Yaskawa INFORM job: X2_104(180,0).JBI

/JOB
//NAME X2_104(180,0)
//POS
///NPOS 390,390,390,11,0,0
///TOOL 0
///POSTYPE PULSE
///PULSE
C00000=2822,-118876,-115474,-188,81202,276
C00001=-104800,-59825,-68378,-15730,82561,27134
C00002=-104796,-59871,-65452,-15790,80804,27361
C00003=-104795,-59835,-64253,-15818,80110,27451
C00004=-104794,-59728,-62536,-15861,79145,27577
C00005=-104795,-59835,-64253,-15818,80110,27451
C00006=-104795,-59821,-63969,-15825,79949,27472
C00007=-104795,-59821,-63967,-15825,79948,27473
C00008=-104795,-59821,-63969,-15825,79949,27472
C00009=-104795,-59821,-63969,-15825,79949,27472
C00010=-104794,-59750,-62822,-15854,79304,27557
C00011=-104793,-59760,-62819,-15854,79297,27558
C00012=-104794,-59750,-62822,-15854,79304,27557
C00013=-104795,-59822,-63970,-15825,79949,27472
C00014=-104795,-59835,-64253,-15818,80110,27451
C00015=-104796,-59871,-65452,-15790,80804,27361
C00016=-104800,-59825,-68378,-15730,82561,27134
C00017=-108679,-64626,-75582,-9628,93281,21595
C00018=-143431,-69229,-73342,20821,87037,-27373
C00019=-148549,-57792,-61137,30779,82601,-29503
C00020=-148549,-57540,-58627,30861,81376,-29834
C00021=-148549,-57408,-57604,30899,80891,-29966
C00022=-148550,-57145,-55796,30970,80047,-30197
C00023=-148549,-57408,-57604,30899,80891,-29966
C00024=-149525,-56700,-57014,31060,81250,-30254
C00025=-148546,-57369,-57388,30906,80793,-29992
C00026=-148548,-57377,-57384,30907,80788,-29994
C00027=-148549,-57379,-57388,30907,80789,-29994
C00028=-148544,-57403,-57724,30893,80955,-29947
C00029=-148544,-57403,-57721,30893,80954,-29947
C00030=-148544,-57403,-57724,30893,80955,-29947
C00031=-148549,-57379,-57388,30907,80789,-29994
C00032=-148549,-57408,-57604,30899,80891,-29966
C00033=-148549,-57540,-58627,30861,81376,-29834
C00034=-148549,-57792,-61137,30779,82601,-29503
C00035=-143431,-69229,-73342,20821,87037,-27373
C00036=-113515,-83541,-80276,-7171,73507,8599
C00037=-114214,-69268,-73638,-6873,76673,8174
C00038=-114213,-69131,-70631,-6922,74904,8274
C00039=-114212,-69024,-69400,-6944,74207,8314
C00040=-114212,-68820,-67637,-6976,73234,8370
C00041=-114212,-69024,-69400,-6944,74207,8314
C00042=-114212,-68905,-68252,-6965,73567,8351
C00043=-114211,-68906,-68249,-6965,73564,8351
C00044=-114212,-68905,-68252,-6965,73567,8351
C00045=-114212,-69039,-69496,-6942,74258,8311
C00046=-114213,-69247,-72540,-6890,76013,8211
C00047=-113515,-83541,-80276,-7171,73507,8599
C00048=-121193,-82756,-80438,381,72886,-91
C00049=-121146,-70418,-74709,362,75701,-66
C00050=-121146,-70284,-71707,364,73922,-71
C00051=-121146,-70176,-70478,365,73221,-73
C00052=-121145,-69975,-68718,367,72241,-76
C00053=-121146,-70176,-70478,365,73221,-73
C00054=-121145,-70029,-69144,367,72475,-75
C00055=-121145,-70029,-69141,367,72474,-75
C00056=-121145,-70029,-69144,367,72475,-75
C00057=-121152,-71796,-70447,369,72370,-78
C00058=-124110,-69926,-69074,1277,72515,-1113
C00059=-138593,-60519,-63927,18922,79598,-16349
C00060=-137648,-60917,-64139,18714,79312,-16056
C00061=-140210,-64003,-66362,19292,79697,-16914
C00062=-130105,-77106,-75700,9072,74443,-7764
C00063=-121203,-87562,-80341,388,70357,-102
C00064=-121146,-70284,-71707,364,73922,-71
C00065=-121146,-70418,-74709,362,75701,-66
C00066=-121193,-82756,-80438,381,72886,-91
C00067=-119439,-80664,-79685,-1380,73580,1904
C00068=-119526,-70071,-74713,-1339,75962,1848
C00069=-119525,-69957,-71718,-1350,74178,1867
C00070=-119525,-69858,-70493,-1354,73475,1875
C00071=-119525,-69668,-68738,-1361,72493,1886
C00072=-119525,-69858,-70493,-1354,73475,1875
C00073=-119525,-69702,-69020,-1360,72649,1884
C00074=-119525,-69702,-69016,-1360,72646,1885
C00075=-119525,-69702,-69020,-1360,72649,1884
C00076=-119525,-69851,-70308,-1355,73364,1876
C00077=-120731,-69912,-70673,-987,73540,1455
C00078=-119525,-69885,-70669,-1354,73569,1874
C00079=-119525,-69895,-70665,-1354,73562,1874
C00080=-119525,-69721,-69012,-1360,72634,1885
C00081=-119525,-69858,-70493,-1354,73475,1875
C00082=-119525,-69957,-71718,-1350,74178,1867
C00083=-119526,-70071,-74713,-1339,75962,1848
C00084=-108249,-94324,-77488,56,64739,4382
C00085=-108596,-86932,-71529,170,64871,4253
C00086=-108725,-84070,-69130,212,64865,4205
C00087=-105542,-82906,-68648,-826,65188,5383
C00088=-119360,-76750,-65885,13584,70522,-11705
C00089=-122073,-72654,-64134,16061,73903,-15414
C00090=-121979,-72766,-64187,16042,73861,-15386
C00091=-122522,-71846,-63747,16636,74615,-16299
C00092=-129432,-59927,-56905,23211,83184,-32001
C00093=-127456,-72696,-62533,22682,75276,-32884
C00094=-129013,-74086,-64315,22925,76062,-33315
C00095=-132460,-77476,-68693,23432,77911,-34241
C00096=-135381,-103003,-79022,24540,72556,-36456
C00097=-155606,-83763,-70294,33424,82257,-10320
C00098=-151405,-68724,-63344,32871,83525,-8251
C00099=-152125,-66994,-60639,32982,83150,-8650
C00100=-148800,-61641,-56056,32604,81881,-7710
C00101=-126757,-81773,-69022,8384,64119,9204
C00102=-127031,-82170,-69267,3063,63090,13556
C00103=-124915,-87939,-73263,2287,62515,14340
C00104=-115381,-93439,-79772,-9030,66985,13175
C00105=-91545,-88698,-72787,-32521,79113,9069
C00106=-71683,-72063,-68966,-26106,87557,15526
C00107=-79934,-51849,-58812,-25261,88765,12201
C00108=-82185,-48076,-53683,-24983,86983,11751
C00109=-83735,-47880,-52547,-24792,85977,11391
C00110=-84464,-48873,-53018,-24699,85557,11210
C00111=-94891,-61855,-60139,-23205,80447,8398
C00112=-100780,-70938,-64689,-19538,73748,2674
C00113=-115179,-76942,-67444,-14121,68125,-4118
C00114=-111498,-78431,-66563,-20592,66506,-6661
C00115=-124355,-85604,-69411,-6892,57492,-20990
C00116=-144608,-76157,-64843,18668,63245,-44599
C00117=-155294,-46121,-48462,31776,84228,-61563
C00118=-157048,-60165,-52454,36767,71330,-65698
C00119=-158808,-60243,-53717,36995,72681,-65990
C00120=-162225,-60657,-56708,37410,75470,-66490
C00121=-167417,-72784,-64632,35375,81907,-66933
C00122=-116272,-113725,-85439,-7807,65506,33606
C00123=-117374,-79868,-72519,-7126,74775,32629
C00124=-119711,-75631,-67242,-6610,73513,31878
C00125=-120783,-73750,-64961,-6368,72993,31529
C00126=-120584,-71036,-63698,-6398,73621,31564
C00127=-120975,-79246,-65174,-5752,61943,44903
C00128=-119928,-81186,-67588,-6116,62507,45272
C00129=-117420,-85347,-72820,-6980,63787,46146
C00130=-116281,-118301,-84670,-8155,54332,47249
C00131=846,-162146,-127518,2443,90805,10094
C00132=846,-162146,-127518,2443,90805,10094
C00133=-127354,-61380,-68788,13702,79975,-24096
C00134=-125311,-61634,-65992,13253,77838,-23621
C00135=-124491,-61652,-64830,13073,76999,-23425
C00136=-124495,-61511,-63095,13123,76029,-23531
C00137=-124491,-61652,-64830,13073,76999,-23425
C00138=-124521,-61630,-64544,13089,76844,-23452
C00139=-124525,-61630,-64553,13090,76850,-23453
C00140=-124521,-61630,-64544,13089,76844,-23452
C00141=-124480,-61634,-64545,13078,76835,-23439
C00142=-124482,-61539,-63385,13111,76187,-23509
C00143=-122660,-61663,-63447,12634,75875,-22900
C00144=-124482,-61539,-63385,13111,76187,-23509
C00145=-124480,-61634,-64545,13078,76835,-23439
C00146=-124491,-61652,-64830,13073,76999,-23425
C00147=-125311,-61634,-65992,13253,77838,-23621
C00148=-127354,-61380,-68788,13702,79975,-24096
C00149=-122646,-60819,-73208,8582,92262,-18154
C00150=-97025,-77240,-76763,-20966,85097,28182
C00151=-93139,-57918,-60776,-30781,82021,29693
C00152=-93133,-57672,-58277,-30872,80802,30026
C00153=-93131,-57543,-57259,-30912,80319,30159
C00154=-93129,-57265,-55441,-30989,79477,30390
C00155=-93131,-57543,-57259,-30912,80319,30159
C00156=-93130,-57513,-57038,-30922,80215,30187
C00157=-93128,-57523,-57046,-30922,80216,30188
C00158=-93130,-57513,-57038,-30922,80215,30187
C00159=-93131,-57509,-57019,-30922,80207,30189
C00160=-93126,-57579,-57367,-30910,80363,30148
C00161=-93126,-57580,-57377,-30909,80367,30147
C00162=-93126,-57579,-57367,-30910,80363,30148
C00163=-93131,-57509,-57019,-30922,80207,30189
C00164=-93131,-57543,-57259,-30912,80319,30159
C00165=-93133,-57672,-58277,-30872,80802,30026
C00166=-93139,-57918,-60776,-30781,82021,29693
C00167=-97025,-77240,-76763,-20966,85097,28182
C00168=-129051,-93674,-83845,7773,70242,-9076
C00169=-127648,-69148,-72931,7145,75952,-8231
C00170=-127649,-68965,-69921,7198,74207,-8333
C00171=-127649,-68840,-68690,7221,73519,-8374
C00172=-127649,-68617,-66917,7256,72550,-8432
C00173=-127649,-68840,-68690,7221,73519,-8374
C00174=-127649,-68692,-67528,7244,72885,-8412
C00175=-127649,-68691,-67535,7244,72890,-8411
C00176=-127649,-68692,-67528,7244,72885,-8412
C00177=-127649,-68843,-68772,7220,73568,-8371
C00178=-127648,-69095,-71818,7164,75299,-8269
C00179=-129051,-93674,-83845,7773,70242,-9076
C00180=-120757,-102453,-87361,-136,66650,45
C00181=-120732,-71973,-74484,-137,74388,45
C00182=-120732,-71738,-71451,-139,72642,47
C00183=-120732,-71593,-70212,-139,71954,48
C00184=-120732,-71339,-68426,-140,70985,49
C00185=-120732,-71593,-70212,-139,71954,48
C00186=-120732,-71405,-68858,-140,71217,48
C00187=-120732,-71406,-68867,-140,71222,48
C00188=-120732,-71405,-68858,-140,71217,48
C00189=-120732,-71373,-68826,-140,71214,48
C00190=-120732,-71507,-69843,-139,71771,48
C00191=-120732,-71519,-69851,-139,71770,48
C00192=-120732,-71507,-69843,-139,71771,48
C00193=-120732,-71601,-70491,-139,72121,47
C00194=-120732,-71593,-70212,-139,71954,48
C00195=-120732,-71738,-71451,-139,72642,47
C00196=-120732,-71973,-74484,-137,74388,45
C00197=-120757,-102453,-87361,-136,66650,45
C00198=-122887,-105945,-88684,1839,65772,-2203
C00199=-122373,-71992,-74562,1588,74513,-1895
C00200=-122373,-71761,-71530,1601,72766,-1918
C00201=-122373,-71617,-70290,1607,72078,-1927
C00202=-122373,-71364,-68505,1615,71109,-1940
C00203=-122373,-71617,-70290,1607,72078,-1927
C00204=-122373,-71408,-68792,1614,71263,-1938
C00205=-122373,-71409,-68799,1614,71267,-1938
C00206=-122373,-71408,-68792,1614,71263,-1938
C00207=-122373,-71581,-70092,1608,71974,-1928
C00208=-122373,-71617,-70466,1606,72186,-1926
C00209=-122373,-71629,-70475,1606,72186,-1926
C00210=-122373,-71617,-70466,1606,72186,-1926
C00211=-122373,-71385,-68772,1614,71263,-1938
C00212=-122373,-71617,-70290,1607,72078,-1927
C00213=-122373,-71761,-71530,1601,72766,-1918
C00214=-122373,-71992,-74562,1588,74513,-1895
C00215=-133268,-95040,-77682,127,64152,-4292
C00216=-132914,-87584,-71736,8,64324,-4160
C00217=-132788,-84746,-69336,-33,64304,-4114
C00218=-135986,-83528,-68799,1028,64630,-5300
C00219=-122065,-77647,-66228,-13513,69975,11894
C00220=-119317,-73595,-64480,-15999,73355,15628
C00221=-119411,-73708,-64532,-15979,73312,15599
C00222=-118527,-72244,-63846,-16799,74509,16993
C00223=-111595,-60993,-57450,-23168,82835,32346
C00224=-113498,-73907,-62961,-22735,74807,33281
C00225=-112101,-75224,-64810,-22943,75622,33648
C00226=-108617,-78641,-69184,-23460,77467,34590
C00227=-104995,-108382,-80828,-24872,71087,37306
C00228=-81107,-97069,-75926,-33957,81080,12730
C00229=-89794,-69286,-63891,-32914,83430,8507
C00230=-92511,-64679,-58817,-32657,81738,7911
C00231=-93502,-63064,-56954,-32563,81088,7703
C00232=-125340,-77919,-68334,6389,68007,-3271
C00233=-122535,-78171,-68492,5506,67769,-2261
C00234=-142571,-65930,-58305,31693,78328,-6211
C00235=-143561,-67945,-60348,31813,78891,-6449
C00236=-146157,-73008,-65581,32111,80403,-7058
C00237=-151976,-96389,-75554,33262,77667,-10217
C00238=-169677,-74631,-70025,26474,86646,-15561
C00239=-161412,-51090,-58299,25576,88476,-12078
C00240=-159165,-47289,-53162,25291,86699,-11632
C00241=-158963,-45086,-50789,25269,86338,-11636
C00242=-158336,-45806,-51137,25187,86007,-11474
C00243=-146793,-61427,-59873,23521,80202,-8401
C00244=-141804,-69475,-63982,20024,73947,-2936
C00245=-126322,-76009,-67109,14276,67996,4203
C00246=-129780,-77698,-66230,20718,66216,6798
C00247=-117038,-85089,-69143,6936,57178,21117
C00248=-96623,-75832,-64695,-18839,63046,44842
C00249=-85691,-45948,-48331,-31884,84166,61886
C00250=-84077,-58564,-51527,-36932,71467,65928
C00251=-82472,-59150,-53149,-37138,72721,66188
C00252=-79083,-59546,-56131,-37554,75503,66675
C00253=-72353,-72252,-64387,-35656,82493,67569
C00254=-120352,-109349,-83964,6698,66011,-31685
C00255=-120416,-78787,-71982,6391,74296,-31254
C00256=-118192,-74362,-66618,5875,73105,-30532
C00257=-117020,-73237,-64754,5602,72455,-30146
C00258=-117327,-69714,-63061,5656,73241,-30219
C00259=-116281,-77938,-64811,4216,61759,-43152
C00260=-117522,-79877,-67041,4686,62176,-43648
C00261=-119910,-84247,-72366,5547,63355,-44498
C00262=-119669,-115920,-83969,5994,54247,-44885
C00263=2000,-115920,-83969,0,54247,0
C00264=2000,-115920,-83969,0,54247,0
C00265=-141550,-97499,-104778,26177,80441,-28547
C00266=-126206,-111975,-82944,22184,64928,-26008
C00267=-122372,-105668,-78021,21264,64116,-24650
C00268=-120931,-103160,-76022,20905,63803,-24139
C00269=-120921,-101974,-73874,21025,63133,-24264
C00270=-120931,-103160,-76022,20905,63803,-24139
C00271=-120951,-102297,-74340,21011,63254,-24252
C00272=-120952,-98942,-73213,20837,64219,-24068
C00273=-120951,-102297,-74340,21011,63254,-24252
C00274=-120814,-100289,-74445,20792,64246,-24008
C00275=-118264,-100229,-74430,20147,63632,-23115
C00276=-120814,-100289,-74445,20792,64246,-24008
C00277=-122217,-102752,-76452,21138,64574,-24500
C00278=-125945,-108938,-81392,22024,65421,-25806
C00279=-120620,-115091,-85499,100,58027,127
C00280=-120625,-106560,-79735,101,58864,125
C00281=-120627,-103290,-77416,101,59118,125
C00282=-120618,-102138,-75286,99,58398,128
C00283=-120627,-103290,-77416,101,59118,125
C00284=-120592,-102634,-75812,89,58467,138
C00285=-120605,-99225,-74663,93,59512,134
C00286=-120592,-102634,-75812,89,58467,138
C00287=-120589,-105878,-78127,88,58225,139
C00288=-120581,-114327,-83877,86,57422,141
C00289=-120609,-115352,-85448,96,57862,131
C00290=-120615,-106812,-79689,97,58706,129
C00291=-120617,-103538,-77372,98,58963,129
C00292=-120608,-102377,-75238,95,58246,132
C00293=-120617,-103538,-77372,98,58963,129
C00294=-120602,-102641,-75605,93,58336,134
C00295=-120615,-99241,-74460,96,59379,130
C00296=-120602,-102641,-75605,93,58336,134
C00297=-120600,-105884,-77920,92,58094,135
C00298=-120593,-114326,-83667,90,57293,137
C00299=-120604,-115480,-85354,94,57738,133
C00300=-120611,-106938,-79599,96,58586,131
C00301=-120613,-103664,-77283,96,58843,130
C00302=-120604,-102497,-75147,94,58128,133
C00303=-120613,-103664,-77283,96,58843,130
C00304=-120606,-102861,-75578,94,58207,132
C00305=-120619,-99464,-74438,98,59251,128
C00306=-120606,-102861,-75578,94,58207,132
C00307=-120604,-106107,-77891,94,57962,133
C00308=-120597,-114556,-83634,92,57154,135
C00309=-120620,-115749,-85311,100,57574,126
C00310=-120626,-107199,-79561,101,58429,125
C00311=-120628,-103920,-77247,102,58689,124
C00312=-120618,-102744,-75107,99,57977,127
C00313=-120628,-103920,-77247,102,58689,124
C00314=-120592,-102876,-75437,89,58112,138
C00315=-120605,-99485,-74300,93,59155,134
C00316=-120592,-102876,-75437,89,58112,138
C00317=-120589,-106121,-77749,89,57868,139
C00318=-120581,-114566,-83489,86,57060,141
C00319=-115079,-112625,-82688,-21971,64604,26312
C00320=-118946,-106323,-77763,-21050,63791,24939
C00321=-120398,-103816,-75763,-20691,63477,24423
C00322=-120389,-102603,-73605,-20815,62818,24552
C00323=-120398,-103816,-75763,-20691,63477,24423
C00324=-120381,-102752,-73855,-20803,62893,24541
C00325=-120401,-99421,-72747,-20622,63854,24351
C00326=-120381,-102752,-73855,-20803,62893,24541
C00327=-117684,-96935,-72649,-22432,67322,27182
C00328=-117673,-92479,-70951,-23618,70462,29315
C00329=-120182,-100632,-73992,-20652,64044,24401
C00330=-118766,-103080,-75998,-20995,64380,24897
C00331=-115003,-109225,-80935,-21875,65246,26214
C00332=-96247,-111176,-86969,-9160,73020,10193
C00333=-97957,-104228,-81170,-8884,72830,9600
C00334=-93225,-110303,-79146,-13824,64256,14788
C00335=-140867,-111118,-79424,-5041,59620,-4980
C00336=-116219,-104435,-72255,-32591,66514,-221
C00337=-115584,-100743,-73698,-31087,72701,-1810
C00338=-113043,-107294,-79247,-31314,73679,-1058
C00339=-144881,-110704,-87119,9425,73387,-9883
C00340=-143181,-103775,-81320,9152,73183,-9295
C00341=-147322,-117161,-79897,15014,57285,-12713
C00342=-91825,-109379,-79334,-3231,60715,9106
C00343=-124930,-105159,-72153,33305,65233,92
C00344=-125516,-100275,-73747,31397,72665,2122
C00345=-128041,-106831,-79296,31633,73644,1375
C00346=-148553,-107836,-85777,9966,74467,-11099
C00347=-146731,-101182,-80016,9692,74121,-10482
C00348=-148903,-108801,-79057,12826,64934,-12232
C00349=-93242,-109245,-79130,-2837,60536,8573
C00350=-94983,-101123,-80123,-55,70977,7714
C00351=-94260,-108369,-86086,-203,70925,7971
C00352=-92903,-107163,-85994,-9620,74852,11237
C00353=-94697,-100547,-80230,-9348,74496,10630
C00354=-90990,-111470,-79091,-14250,61612,13428
C00355=-148758,-109871,-79037,3193,59655,-8641
C00356=-153240,-110220,-78573,5727,58282,-10530
C00357=-146194,-101027,-80277,310,71255,-7446
C00358=-146914,-108261,-86241,457,71212,-7702
C00359=-146914,-110318,-91010,453,73090,-7695
C00360=-146914,-110318,-91010,453,73090,-7695
C00361=-128621,-115405,-83679,-32201,62902,1684
C00362=-109158,-114787,-67564,-57970,59113,29930
C00363=-123032,-111080,-63821,-57176,47551,25820
C00364=-123402,-108210,-57218,-59198,45926,27093
C00365=-132906,-111039,-65804,-41029,44976,19022
C00366=-130912,-121589,-79027,-33705,49955,17163
C00367=-130912,-127210,-87126,-32783,51722,16500
C00368=-111497,-99476,-74625,-44606,72972,57685
C00369=-143951,-87931,-76629,-13326,69430,45386
C00370=-142667,-81717,-73015,-13610,70590,45724
C00371=-141368,-75160,-69101,-13897,71741,46063
C00372=-139856,-91310,-81083,-14385,71107,46692
C00373=-147106,-116431,-118144,4230,76181,-7502
C00374=-101608,-95614,-84790,8586,63966,9623
C00375=-106266,-75316,-61399,29605,53199,-18730
C00376=-98654,-69900,-56335,21783,48246,-12977
C00377=-97773,-68120,-54602,21305,47872,-12642
C00378=-97613,-69374,-54502,21441,47172,-12733
C00379=-96912,-68892,-50244,21842,44775,-12972
C00380=-92902,-55713,-51680,10842,62710,-8765
C00381=-97147,-68860,-63059,12526,63566,-10301
C00382=-100017,-32969,-51929,13447,85098,-38502
C00383=-91186,-27541,-47207,3454,85632,-36582
C00384=-94361,-22653,-42642,7012,85824,-37196
C00385=-96330,-17023,-36235,8317,83572,-37915
C00386=-103618,-23212,-42014,14317,84633,-39771
C00387=-111426,-38573,-59092,16054,88569,-41926
C00388=-147106,-116431,-118144,4230,76181,-7502
C00389=2000,-115920,-83969,0,54247,0
BC00000=0,666204,878766
BC00001=23900,723356,53
BC00002=20311,727498,53
BC00003=18875,729154,53
BC00004=18891,729150,53
BC00005=18875,729154,53
BC00006=18925,729694,53
BC00007=18917,732766,53
BC00008=18925,729694,53
BC00009=18857,729153,53
BC00010=18868,729174,53
BC00011=15682,729167,53
BC00012=18868,729174,53
BC00013=18857,729153,53
BC00014=18875,729154,53
BC00015=20311,727498,53
BC00016=23900,723356,53
BC00017=22934,724458,53
BC00018=74464,724323,53
BC00019=73591,723467,53
BC00020=78215,727921,53
BC00021=80065,729702,53
BC00022=80081,729698,53
BC00023=80065,729702,53
BC00024=80582,729701,53
BC00025=83767,729709,53
BC00026=80582,729701,53
BC00027=80082,724004,53
BC00028=87416,724022,53
BC00029=87408,727094,53
BC00030=87416,724022,53
BC00031=80082,724004,53
BC00032=80065,729702,53
BC00033=78215,727921,53
BC00034=73591,723467,53
BC00035=74464,724323,53
BC00036=129427,721333,53
BC00037=129427,721333,53
BC00038=128190,726618,53
BC00039=127695,728732,53
BC00040=127711,728728,53
BC00041=127695,728732,53
BC00042=125403,727840,53
BC00043=124687,730834,53
BC00044=125403,727840,53
BC00045=125897,725726,53
BC00046=127135,720441,53
BC00047=129427,721333,53
BC00048=333799,722934,53
BC00049=333799,722934,53
BC00050=333814,728358,53
BC00051=333819,730528,53
BC00052=333836,730524,53
BC00053=333819,730528,53
BC00054=333841,730600,53
BC00055=333833,733673,53
BC00056=333841,730600,53
BC00057=325529,727454,53
BC00058=325529,727454,53
BC00059=322627,730075,53
BC00060=322627,730075,53
BC00061=322627,730075,53
BC00062=324335,729077,53
BC00063=333819,730528,53
BC00064=333814,728358,53
BC00065=333799,722934,53
BC00066=333799,722934,53
BC00067=390689,722481,53
BC00068=390689,722481,53
BC00069=390412,727894,53
BC00070=390301,730059,53
BC00071=390317,730055,53
BC00072=390301,730059,53
BC00073=390304,730021,53
BC00074=390131,733088,53
BC00075=390304,730021,53
BC00076=387191,728800,53
BC00077=383848,732963,53
BC00078=387029,733130,53
BC00079=383848,732963,53
BC00080=384046,729728,53
BC00081=390301,730059,53
BC00082=390412,727894,53
BC00083=390689,722481,53
BC00084=362376,748394,38812
BC00085=362376,748394,38812
BC00086=362376,748394,38812
BC00087=362376,748394,38812
BC00088=362376,748394,38812
BC00089=362376,748394,38812
BC00090=362376,748394,38812
BC00091=362376,748394,38812
BC00092=362376,748394,38812
BC00093=362376,748394,38812
BC00094=362376,748394,38812
BC00095=362376,748394,38812
BC00096=362376,748394,38812
BC00097=337816,741481,25289
BC00098=337816,741481,25289
BC00099=337816,741481,25289
BC00100=337817,741482,25288
BC00101=337817,741482,25288
BC00102=337817,741482,25288
BC00103=337817,741482,25288
BC00104=337817,741482,25288
BC00105=337816,741481,25289
BC00106=96213,735243,20905
BC00107=97498,733107,17680
BC00108=97498,733107,17680
BC00109=97498,733107,17680
BC00110=97498,733107,17680
BC00111=97498,733107,17680
BC00112=97498,733107,17680
BC00113=97498,733107,17680
BC00114=97498,733107,17680
BC00115=97498,733107,17680
BC00116=97498,733107,17680
BC00117=97498,733107,17680
BC00118=97498,733107,17680
BC00119=97498,733107,17680
BC00120=97498,733107,17680
BC00121=96213,735243,20905
BC00122=34912,743660,44528
BC00123=34912,743660,44528
BC00124=34912,743660,44528
BC00125=34912,743660,44528
BC00126=34912,743660,44528
BC00127=34912,743660,44528
BC00128=34912,743660,44528
BC00129=34912,743660,44528
BC00130=34912,743660,44528
BC00131=225332,668039,21215
BC00132=225332,668039,21215
BC00133=398174,724912,53
BC00134=398174,729107,53
BC00135=398174,730785,53
BC00136=398174,730802,53
BC00137=398174,730785,53
BC00138=398174,731328,53
BC00139=398174,734400,53
BC00140=398174,731328,53
BC00141=398174,730788,53
BC00142=398174,730822,53
BC00143=398174,730830,53
BC00144=398174,730822,53
BC00145=398174,730788,53
BC00146=398174,730785,53
BC00147=398174,729107,53
BC00148=398174,724912,53
BC00149=398174,726011,53
BC00150=364496,725635,53
BC00151=365379,724793,53
BC00152=360747,729255,53
BC00153=358894,731039,53
BC00154=358889,731056,53
BC00155=358894,731039,53
BC00156=358379,731038,53
BC00157=355194,731030,53
BC00158=358379,731038,53
BC00159=358908,725343,53
BC00160=351572,725322,53
BC00161=351564,728394,53
BC00162=351572,725322,53
BC00163=358908,725343,53
BC00164=358894,731039,53
BC00165=360747,729255,53
BC00166=365379,724793,53
BC00167=364496,725635,53
BC00168=309549,722382,53
BC00169=309549,722382,53
BC00170=310778,727709,53
BC00171=311269,729840,53
BC00172=311264,729857,53
BC00173=311269,729840,53
BC00174=313573,728972,53
BC00175=314274,731969,53
BC00176=313573,728972,53
BC00177=313082,726841,53
BC00178=311853,721514,53
BC00179=309549,722382,53
BC00180=105169,723000,53
BC00181=105169,723000,53
BC00182=105145,728460,53
BC00183=105136,730644,53
BC00184=105130,730660,53
BC00185=105136,730644,53
BC00186=105122,730732,53
BC00187=105114,733804,53
BC00188=105122,730732,53
BC00189=113450,727626,53
BC00190=116706,730590,53
BC00191=113521,730583,53
BC00192=116706,730590,53
BC00193=113358,728488,53
BC00194=105136,730644,53
BC00195=105145,728460,53
BC00196=105169,723000,53
BC00197=105169,723000,53
BC00198=48282,722274,53
BC00199=48282,722274,53
BC00200=48550,727724,53
BC00201=48657,729904,53
BC00202=48651,729921,53
BC00203=48657,729904,53
BC00204=48663,729883,53
BC00205=48820,732951,53
BC00206=48663,729883,53
BC00207=51775,728662,53
BC00208=55093,732837,53
BC00209=51912,732988,53
BC00210=55093,732837,53
BC00211=54923,729620,53
BC00212=48657,729904,53
BC00213=48550,727724,53
BC00214=48282,722274,53
BC00215=75858,747378,32664
BC00216=75858,747378,32664
BC00217=75858,747378,32664
BC00218=75858,747378,32664
BC00219=75858,747378,32664
BC00220=75858,747378,32664
BC00221=75858,747378,32664
BC00222=75858,747378,32664
BC00223=75858,747378,32664
BC00224=75858,747378,32664
BC00225=75858,747378,32664
BC00226=75858,747378,32664
BC00227=75858,747378,32664
BC00228=100335,741000,19110
BC00229=100335,741000,19110
BC00230=100335,741000,19110
BC00231=100335,741000,19110
BC00232=100335,741000,19110
BC00233=100335,741000,19110
BC00234=100335,741000,19110
BC00235=100335,741000,19110
BC00236=100335,741000,19110
BC00237=100335,741000,19110
BC00238=340452,735599,16827
BC00239=340990,733472,13046
BC00240=340990,733472,13046
BC00241=340990,733472,13046
BC00242=340990,733472,13046
BC00243=340990,733472,13046
BC00244=340990,733472,13046
BC00245=340990,733472,13046
BC00246=340990,733472,13046
BC00247=340990,733472,13046
BC00248=340990,733472,13046
BC00249=340990,733472,13046
BC00250=340990,733472,13046
BC00251=340990,733472,13046
BC00252=340990,733472,13046
BC00253=340452,735599,16827
BC00254=398174,745222,42722
BC00255=398174,745222,42722
BC00256=398174,745222,42722
BC00257=398174,745222,42722
BC00258=398174,745222,42722
BC00259=398174,745222,42722
BC00260=398174,745222,42722
BC00261=398174,745222,42722
BC00262=398174,745222,42722
BC00263=262890,666204,990547
BC00264=262890,666204,990547
BC00265=337114,755302,1075175
BC00266=337114,800894,1075175
BC00267=337114,800894,1075175
BC00268=337114,800894,1075175
BC00269=337114,800894,1075175
BC00270=337114,800894,1075175
BC00271=337114,800894,1075175
BC00272=337114,800894,1075175
BC00273=337114,800894,1075175
BC00274=337114,800894,1075175
BC00275=337114,800894,1075175
BC00276=337114,800894,1075175
BC00277=337114,800894,1075175
BC00278=337114,800894,1075175
BC00279=314961,788371,1075175
BC00280=314961,788371,1075175
BC00281=314961,788371,1075175
BC00282=314961,788371,1075175
BC00283=314961,788371,1075175
BC00284=314961,788371,1075175
BC00285=314961,788371,1075175
BC00286=314961,788371,1075175
BC00287=314961,788371,1075175
BC00288=314961,788371,1075175
BC00289=250925,788006,1075175
BC00290=250925,788006,1075175
BC00291=250925,788006,1075175
BC00292=250925,788006,1075175
BC00293=250925,788006,1075175
BC00294=250925,788006,1075175
BC00295=250925,788006,1075175
BC00296=250925,788006,1075175
BC00297=250925,788006,1075175
BC00298=250925,788006,1075175
BC00299=182224,787817,1075175
BC00300=182224,787817,1075175
BC00301=182224,787817,1075175
BC00302=182224,787817,1075175
BC00303=182224,787817,1075175
BC00304=182224,787817,1075175
BC00305=182224,787817,1075175
BC00306=182224,787817,1075175
BC00307=182224,787817,1075175
BC00308=182224,787817,1075175
BC00309=121128,787483,1075175
BC00310=121128,787483,1075175
BC00311=121128,787483,1075175
BC00312=121128,787483,1075175
BC00313=121128,787483,1075175
BC00314=121128,787483,1075175
BC00315=121128,787483,1075175
BC00316=121128,787483,1075175
BC00317=121128,787483,1075175
BC00318=121128,787483,1075175
BC00319=98740,799429,1075175
BC00320=98740,799429,1075175
BC00321=98740,799429,1075175
BC00322=98740,799429,1075175
BC00323=98740,799429,1075175
BC00324=98740,799429,1075175
BC00325=98740,799429,1075175
BC00326=98740,799429,1075175
BC00327=98740,799429,1075175
BC00328=98740,799429,1075175
BC00329=98740,799429,1075175
BC00330=98740,799429,1075175
BC00331=98740,799429,1075175
BC00332=103096,808765,1075175
BC00333=103096,808765,1075175
BC00334=103096,808765,1075175
BC00335=103096,808765,1075175
BC00336=103096,808765,1075175
BC00337=103096,808765,1075175
BC00338=103096,808765,1075175
BC00339=332893,809568,1075175
BC00340=332893,809568,1075175
BC00341=332893,809568,1075175
BC00342=332893,809568,1075175
BC00343=332893,809568,1075175
BC00344=332893,809568,1075175
BC00345=332893,809568,1075175
BC00346=143959,807707,1075175
BC00347=143959,807707,1075175
BC00348=143959,807707,1075175
BC00349=143959,807707,1075175
BC00350=143959,807707,1075175
BC00351=143959,807707,1075175
BC00352=291971,808199,1075175
BC00353=291971,808199,1075175
BC00354=291971,808199,1075175
BC00355=291971,808199,1075175
BC00356=291971,808199,1075175
BC00357=291971,808199,1075175
BC00358=291971,808199,1075175
BC00359=291971,808199,1075175
BC00360=130958,808199,1075175
BC00361=130958,808199,1075175
BC00362=130958,808199,1075175
BC00363=130958,808199,1075175
BC00364=130958,808199,1075175
BC00365=130958,808199,1075175
BC00366=130958,808199,1075175
BC00367=130958,808199,1075175
BC00368=130958,808199,1075175
BC00369=130958,808199,1075175
BC00370=130958,808199,1075175
BC00371=130958,808199,1075175
BC00372=130958,808199,1075175
BC00373=291971,760262,1075175
BC00374=290727,760633,1075175
BC00375=290727,760633,1075175
BC00376=290727,760633,1075175
BC00377=290727,760633,1075175
BC00378=290727,760633,1075175
BC00379=290727,760633,1075175
BC00380=290727,760633,1075175
BC00381=290727,760633,1075175
BC00382=290728,760632,1075172
BC00383=290728,760632,1075172
BC00384=290728,760632,1075172
BC00385=290728,760632,1075172
BC00386=290728,760632,1075172
BC00387=290728,760632,1075172
BC00388=291971,760262,1075175
BC00389=262890,666204,990547
EC00000=1596313,0
EC00001=1596313,0
EC00002=1596313,0
EC00003=1596313,0
EC00004=1596313,0
EC00005=1596313,0
EC00006=1596313,0
EC00007=1596313,0
EC00008=1596313,0
EC00009=1596313,0
EC00010=1596313,0
EC00011=1596313,0
EC00012=1596313,0
EC00013=1596313,0
EC00014=1596313,0
EC00015=1596313,0
EC00016=1596313,0
EC00017=1596313,0
EC00018=1596313,0
EC00019=1596313,0
EC00020=1596313,0
EC00021=1596313,0
EC00022=1596313,0
EC00023=1596313,0
EC00024=1596313,0
EC00025=1596313,0
EC00026=1596313,0
EC00027=1596313,0
EC00028=1596313,0
EC00029=1596313,0
EC00030=1596313,0
EC00031=1596313,0
EC00032=1596313,0
EC00033=1596313,0
EC00034=1596313,0
EC00035=1596313,0
EC00036=1596313,0
EC00037=1596313,0
EC00038=1596313,0
EC00039=1596313,0
EC00040=1596313,0
EC00041=1596313,0
EC00042=1596313,0
EC00043=1596313,0
EC00044=1596313,0
EC00045=1596313,0
EC00046=1596313,0
EC00047=1596313,0
EC00048=1596313,0
EC00049=1596313,0
EC00050=1596313,0
EC00051=1596313,0
EC00052=1596313,0
EC00053=1596313,0
EC00054=1596313,0
EC00055=1596313,0
EC00056=1596313,0
EC00057=1596313,0
EC00058=1596313,0
EC00059=1596313,0
EC00060=1596313,0
EC00061=1596313,0
EC00062=1596313,0
EC00063=1596313,0
EC00064=1596313,0
EC00065=1596313,0
EC00066=1596313,0
EC00067=1596313,0
EC00068=1596313,0
EC00069=1596313,0
EC00070=1596313,0
EC00071=1596313,0
EC00072=1596313,0
EC00073=1596313,0
EC00074=1596313,0
EC00075=1596313,0
EC00076=1596313,0
EC00077=1596313,0
EC00078=1596313,0
EC00079=1596313,0
EC00080=1596313,0
EC00081=1596313,0
EC00082=1596313,0
EC00083=1596313,0
EC00084=1596313,0
EC00085=1596313,0
EC00086=1596313,0
EC00087=1596313,0
EC00088=1596313,0
EC00089=1596313,0
EC00090=1596313,0
EC00091=1596313,0
EC00092=1596313,0
EC00093=1596313,0
EC00094=1596313,0
EC00095=1596313,0
EC00096=1596313,0
EC00097=1596313,0
EC00098=1596313,0
EC00099=1596313,0
EC00100=1596312,0
EC00101=1596312,0
EC00102=1596312,0
EC00103=1596312,0
EC00104=1596312,0
EC00105=1596313,0
EC00106=1596313,0
EC00107=1596313,0
EC00108=1596313,0
EC00109=1596313,0
EC00110=1596313,0
EC00111=1596313,0
EC00112=1596313,0
EC00113=1596313,0
EC00114=1596313,0
EC00115=1596313,0
EC00116=1596313,0
EC00117=1596313,0
EC00118=1596313,0
EC00119=1596313,0
EC00120=1596313,0
EC00121=1596313,0
EC00122=1596313,0
EC00123=1596313,0
EC00124=1596313,0
EC00125=1596313,0
EC00126=1596313,0
EC00127=1596313,0
EC00128=1596313,0
EC00129=1596313,0
EC00130=1596313,0
EC00131=1596313,0
EC00132=1596313,1112951
EC00133=1596313,1112951
EC00134=1596313,1112951
EC00135=1596313,1112951
EC00136=1596313,1112951
EC00137=1596313,1112951
EC00138=1596313,1112951
EC00139=1596313,1112951
EC00140=1596313,1112951
EC00141=1596313,1112951
EC00142=1596313,1112951
EC00143=1596313,1112951
EC00144=1596313,1112951
EC00145=1596313,1112951
EC00146=1596313,1112951
EC00147=1596313,1112951
EC00148=1596313,1112951
EC00149=1596313,1112951
EC00150=1596313,1112951
EC00151=1596313,1112951
EC00152=1596313,1112951
EC00153=1596313,1112951
EC00154=1596313,1112951
EC00155=1596313,1112951
EC00156=1596313,1112951
EC00157=1596313,1112951
EC00158=1596313,1112951
EC00159=1596313,1112951
EC00160=1596313,1112951
EC00161=1596313,1112951
EC00162=1596313,1112951
EC00163=1596313,1112951
EC00164=1596313,1112951
EC00165=1596313,1112951
EC00166=1596313,1112951
EC00167=1596313,1112951
EC00168=1596313,1112951
EC00169=1596313,1112951
EC00170=1596313,1112951
EC00171=1596313,1112951
EC00172=1596313,1112951
EC00173=1596313,1112951
EC00174=1596313,1112951
EC00175=1596313,1112951
EC00176=1596313,1112951
EC00177=1596313,1112951
EC00178=1596313,1112951
EC00179=1596313,1112951
EC00180=1596313,1112951
EC00181=1596313,1112951
EC00182=1596313,1112951
EC00183=1596313,1112951
EC00184=1596313,1112951
EC00185=1596313,1112951
EC00186=1596313,1112951
EC00187=1596313,1112951
EC00188=1596313,1112951
EC00189=1596313,1112951
EC00190=1596313,1112951
EC00191=1596313,1112951
EC00192=1596313,1112951
EC00193=1596313,1112951
EC00194=1596313,1112951
EC00195=1596313,1112951
EC00196=1596313,1112951
EC00197=1596313,1112951
EC00198=1596313,1112951
EC00199=1596313,1112951
EC00200=1596313,1112951
EC00201=1596313,1112951
EC00202=1596313,1112951
EC00203=1596313,1112951
EC00204=1596313,1112951
EC00205=1596313,1112951
EC00206=1596313,1112951
EC00207=1596313,1112951
EC00208=1596313,1112951
EC00209=1596313,1112951
EC00210=1596313,1112951
EC00211=1596313,1112951
EC00212=1596313,1112951
EC00213=1596313,1112951
EC00214=1596313,1112951
EC00215=1596313,1112951
EC00216=1596313,1112951
EC00217=1596313,1112951
EC00218=1596313,1112951
EC00219=1596313,1112951
EC00220=1596313,1112951
EC00221=1596313,1112951
EC00222=1596313,1112951
EC00223=1596313,1112951
EC00224=1596313,1112951
EC00225=1596313,1112951
EC00226=1596313,1112951
EC00227=1596313,1112951
EC00228=1596313,1112951
EC00229=1596313,1112951
EC00230=1596313,1112951
EC00231=1596313,1112951
EC00232=1596313,1112951
EC00233=1596313,1112951
EC00234=1596313,1112951
EC00235=1596313,1112951
EC00236=1596313,1112951
EC00237=1596313,1112951
EC00238=1596313,1112951
EC00239=1596313,1112951
EC00240=1596313,1112951
EC00241=1596313,1112951
EC00242=1596313,1112951
EC00243=1596313,1112951
EC00244=1596313,1112951
EC00245=1596313,1112951
EC00246=1596313,1112951
EC00247=1596313,1112951
EC00248=1596313,1112951
EC00249=1596313,1112951
EC00250=1596313,1112951
EC00251=1596313,1112951
EC00252=1596313,1112951
EC00253=1596313,1112951
EC00254=1596313,1112951
EC00255=1596313,1112951
EC00256=1596313,1112951
EC00257=1596313,1112951
EC00258=1596313,1112951
EC00259=1596313,1112951
EC00260=1596313,1112951
EC00261=1596313,1112951
EC00262=1596313,1112951
EC00263=1596313,1112951
EC00264=1596313,-556475
EC00265=1330261,-556475
EC00266=1330261,-556475
EC00267=1330261,-556475
EC00268=1330261,-556475
EC00269=1330261,-556475
EC00270=1330261,-556475
EC00271=1330261,-556475
EC00272=1330261,-556475
EC00273=1330261,-556475
EC00274=1330261,-556475
EC00275=1330261,-556475
EC00276=1330261,-556475
EC00277=1330261,-556475
EC00278=1330261,-556475
EC00279=1330261,-556475
EC00280=1330261,-556475
EC00281=1330261,-556475
EC00282=1330261,-556475
EC00283=1330261,-556475
EC00284=1330261,-556475
EC00285=1330261,-556475
EC00286=1330261,-556475
EC00287=1330261,-556475
EC00288=1330261,-556475
EC00289=1330261,-556475
EC00290=1330261,-556475
EC00291=1330261,-556475
EC00292=1330261,-556475
EC00293=1330261,-556475
EC00294=1330261,-556475
EC00295=1330261,-556475
EC00296=1330261,-556475
EC00297=1330261,-556475
EC00298=1330261,-556475
EC00299=1330261,-556475
EC00300=1330261,-556475
EC00301=1330261,-556475
EC00302=1330261,-556475
EC00303=1330261,-556475
EC00304=1330261,-556475
EC00305=1330261,-556475
EC00306=1330261,-556475
EC00307=1330261,-556475
EC00308=1330261,-556475
EC00309=1330261,-556475
EC00310=1330261,-556475
EC00311=1330261,-556475
EC00312=1330261,-556475
EC00313=1330261,-556475
EC00314=1330261,-556475
EC00315=1330261,-556475
EC00316=1330261,-556475
EC00317=1330261,-556475
EC00318=1330261,-556475
EC00319=1330261,-556475
EC00320=1330261,-556475
EC00321=1330261,-556475
EC00322=1330261,-556475
EC00323=1330261,-556475
EC00324=1330261,-556475
EC00325=1330261,-556475
EC00326=1330261,-556475
EC00327=1330261,-556475
EC00328=1330261,-556475
EC00329=1330261,-556475
EC00330=1330261,-556475
EC00331=1330261,-556475
EC00332=1330261,-556475
EC00333=1330261,-556475
EC00334=1330261,-556475
EC00335=1330261,-556475
EC00336=1330261,-556475
EC00337=1330261,-556475
EC00338=1330261,-556475
EC00339=1330261,-556475
EC00340=1330261,-556475
EC00341=1330261,-556475
EC00342=1330261,-556475
EC00343=1330261,-556475
EC00344=1330261,-556475
EC00345=1330261,-556475
EC00346=1330261,-556475
EC00347=1330261,-556475
EC00348=1330261,-556475
EC00349=1330261,-556475
EC00350=1330261,-556475
EC00351=1330261,-556475
EC00352=1330261,-556475
EC00353=1330261,-556475
EC00354=1330261,-556475
EC00355=1330261,-556475
EC00356=1330261,-556475
EC00357=1330261,-556475
EC00358=1330261,-556475
EC00359=1330261,-556475
EC00360=1330261,-556475
EC00361=1330261,-556475
EC00362=1330261,-556475
EC00363=1330261,-556475
EC00364=1330261,-556475
EC00365=1330261,-556475
EC00366=1330261,-556475
EC00367=1330261,-556475
EC00368=1330261,-556475
EC00369=1330261,-556475
EC00370=1330261,-556475
EC00371=1330261,-556475
EC00372=1330261,-556475
EC00373=1330261,-556475
EC00374=1330261,-556475
EC00375=1330261,-556475
EC00376=1330261,-556475
EC00377=1330261,-556475
EC00378=1330261,-556475
EC00379=1330261,-556475
EC00380=1330261,-556475
EC00381=1330261,-556475
EC00382=1330262,-556475
EC00383=1330262,-556475
EC00384=1330262,-556475
EC00385=1330262,-556475
EC00386=1330262,-556475
EC00387=1330262,-556475
EC00388=1330261,-556475
EC00389=1596313,-556475
///POSTYPE BASE
///RECTAN
///RCONF 0,0,0,0,0,0,0,0,0,0,0,0,0,0,0,0,0,0,0,0,0,0,0,0
P00006=0.222,-3.123,-1.508,0.0000,0.0000,0.0000
P00021=-0.225,-6.128,-0.405,0.0000,0.0000,0.0000
P00022=0.222,-3.123,-1.508,0.0000,0.0000,0.0000
P00023=0.143,-0.036,0.682,0.0000,0.0000,0.0000
P00024=0.145,-0.552,1.326,0.0000,0.0000,0.0000
P00025=-2.003,0.006,0.728,0.0000,0.0000,0.0000
P00031=1.853,-0.001,-1.549,0.0000,0.0000,0.0000
P00032=1.957,0.503,-7.217,0.0000,0.0000,0.0000
///RCONF 0,0,0,0,1,0,0,0,0,0,0,0,0,0,0,0,0,0,0,0,0,0,0,0
P00033=-0.123,0.612,-5.012,0.0000,0.0000,0.0000
///RCONF 0,0,0,0,0,0,0,0,0,0,0,0,0,0,0,0,0,0,0,0,0,0,0,0
P00034=-0.304,0.773,-2.693,0.0000,0.0000,0.0000
P00035=2.817,0.591,-1.622,0.0000,0.0000,0.0000
//INST
///DATE 2024/10/31 09:55
///ATTR SC,RW
///GROUP1 RB1,BS1
///GROUP2 ST1
NOP
'X2_104(180,0)
MOVJ C00000 BC00000 VJ=100.00  +MOVJ EC00000 VJ=100.00
'Path S4732
SFTOF3D
MOVJ C00001 BC00001 VJ=100.00  +MOVJ EC00001 VJ=100.00
MOVL C00002 BC00002 V=800.0  +MOVJ EC00002 VJ=100.00
SMOVL C00003 BC00003 V=166.7  +MOVJ EC00003
SREFP 3 C00004 BC00004  +REFP EC00004
CALL JOB:SEARCH-R1-S13D
SET P025 P006
SFTON3D P025
SMOVL C00005 BC00005 V=166.7  +MOVJ EC00005
SMOVL C00006 BC00006 V=166.7  +MOVJ EC00006
SREFP 3 C00007 BC00007  +REFP EC00007
CALL JOB:SEARCH-R1-S13D
SET P025 P006
SFTON3D P025
SMOVL C00008 BC00008 V=166.7  +MOVJ EC00008
SMOVL C00009 BC00009 V=166.7  +MOVJ EC00009
SMOVL C00010 BC00010 V=166.7  +MOVJ EC00010
SREFP 3 C00011 BC00011  +REFP EC00011
CALL JOB:SEARCH-R1-S13D
SET P025 P006
SFTON3D P025
SMOVL C00012 BC00012 V=166.7  +MOVJ EC00012
SMOVL C00013 BC00013 V=166.7  +MOVJ EC00013
SMOVL C00014 BC00014 V=166.7  +MOVJ EC00014
MOVL C00015 BC00015 V=800.0  +MOVJ EC00015 VJ=100.00
MOVL C00016 BC00016 V=1000.0  +MOVJ EC00016 VJ=100.00
'EndPath S4732
MOVJ C00017 BC00017 VJ=100.00  +MOVJ EC00017 VJ=100.00
MOVJ C00018 BC00018 VJ=100.00  +MOVJ EC00018 VJ=100.00
'Path S4733
SFTOF3D
MOVJ C00019 BC00019 VJ=100.00  +MOVJ EC00019 VJ=100.00
MOVL C00020 BC00020 V=800.0  +MOVJ EC00020 VJ=100.00
SMOVL C00021 BC00021 V=166.7  +MOVJ EC00021
SREFP 3 C00022 BC00022  +REFP EC00022
CALL JOB:SEARCH-R1-S13D
SET P024 P006
SFTON3D P024
SMOVL C00023 BC00023 V=166.7  +MOVJ EC00023
SMOVL C00024 BC00024 V=166.7  +MOVJ EC00024
SREFP 3 C00025 BC00025  +REFP EC00025
CALL JOB:SEARCH-R1-S13D
SET P024 P006
SFTON3D P024
SMOVL C00026 BC00026 V=166.7  +MOVJ EC00026
SMOVL C00027 BC00027 V=166.7  +MOVJ EC00027
SMOVL C00028 BC00028 V=166.7  +MOVJ EC00028
SREFP 3 C00029 BC00029  +REFP EC00029
CALL JOB:SEARCH-R1-S13D
SET P024 P006
SFTON3D P024
SMOVL C00030 BC00030 V=166.7  +MOVJ EC00030
SMOVL C00031 BC00031 V=166.7  +MOVJ EC00031
SMOVL C00032 BC00032 V=166.7  +MOVJ EC00032
MOVL C00033 BC00033 V=800.0  +MOVJ EC00033 VJ=100.00
MOVL C00034 BC00034 V=1000.0  +MOVJ EC00034 VJ=100.00
'EndPath S4733
MOVJ C00035 BC00035 VJ=100.00  +MOVJ EC00035 VJ=100.00
MOVJ C00036 BC00036 VJ=100.00  +MOVJ EC00036 VJ=100.00
'Path S4734
SFTOF3D
MOVJ C00037 BC00037 VJ=100.00  +MOVJ EC00037 VJ=100.00
MOVL C00038 BC00038 V=800.0  +MOVJ EC00038 VJ=100.00
SMOVL C00039 BC00039 V=166.7  +MOVJ EC00039
SREFP 3 C00040 BC00040  +REFP EC00040
CALL JOB:SEARCH-R1-S13D
SET P023 P006
SFTON3D P023
SMOVL C00041 BC00041 V=166.7  +MOVJ EC00041
SMOVL C00042 BC00042 V=166.7  +MOVJ EC00042
SREFP 3 C00043 BC00043  +REFP EC00043
CALL JOB:SEARCH-R1-S13D
SET P023 P006
SFTON3D P023
SMOVL C00044 BC00044 V=166.7  +MOVJ EC00044
MOVL C00045 BC00045 V=800.0  +MOVJ EC00045 VJ=100.00
MOVL C00046 BC00046 V=1000.0  +MOVJ EC00046 VJ=100.00
'EndPath S4734
MOVJ C00047 BC00047 VJ=100.00  +MOVJ EC00047 VJ=100.00
MOVJ C00048 BC00048 VJ=100.00  +MOVJ EC00048 VJ=100.00
'Path S4735
SFTOF3D
MOVJ C00049 BC00049 VJ=100.00  +MOVJ EC00049 VJ=100.00
MOVL C00050 BC00050 V=800.0  +MOVJ EC00050 VJ=100.00
SMOVL C00051 BC00051 V=166.7  +MOVJ EC00051
SREFP 3 C00052 BC00052  +REFP EC00052
CALL JOB:SEARCH-R1-S13D
SET P022 P006
SFTON3D P022
SMOVL C00053 BC00053 V=166.7  +MOVJ EC00053
SMOVL C00054 BC00054 V=166.7  +MOVJ EC00054
SREFP 3 C00055 BC00055  +REFP EC00055
CALL JOB:SEARCH-R1-S13D
SET P022 P006
SFTON3D P022
SMOVL C00056 BC00056 V=166.7  +MOVJ EC00056
SMOVL C00057 BC00057 V=166.7  +MOVJ EC00057
SMOVL C00058 BC00058 V=133.3  +MOVJ EC00058
SMOVL C00059 BC00059 V=166.7  +MOVJ EC00059
SREFP 3 C00060 BC00060  +REFP EC00060
CALL JOB:SEARCH-R1-S13D
SET P022 P006
SFTON3D P022
SMOVL C00061 BC00061 V=166.7  +MOVJ EC00061
SMOVL C00062 BC00062 V=166.7  +MOVJ EC00062
SMOVL C00063 BC00063 V=166.7  +MOVJ EC00063
MOVL C00064 BC00064 V=800.0  +MOVJ EC00064 VJ=100.00
MOVL C00065 BC00065 V=1000.0  +MOVJ EC00065 VJ=100.00
'EndPath S4735
MOVJ C00066 BC00066 VJ=100.00  +MOVJ EC00066 VJ=100.00
MOVJ C00067 BC00067 VJ=100.00  +MOVJ EC00067 VJ=100.00
'Path S4736
SFTOF3D
MOVJ C00068 BC00068 VJ=100.00  +MOVJ EC00068 VJ=100.00
MOVL C00069 BC00069 V=800.0  +MOVJ EC00069 VJ=100.00
SMOVL C00070 BC00070 V=166.7  +MOVJ EC00070
SREFP 3 C00071 BC00071  +REFP EC00071
CALL JOB:SEARCH-R1-S13D
SET P021 P006
SFTON3D P021
SMOVL C00072 BC00072 V=166.7  +MOVJ EC00072
SMOVL C00073 BC00073 V=166.7  +MOVJ EC00073
SREFP 3 C00074 BC00074  +REFP EC00074
CALL JOB:SEARCH-R1-S13D
SET P021 P006
SFTON3D P021
SMOVL C00075 BC00075 V=166.7  +MOVJ EC00075
SMOVL C00076 BC00076 V=166.7  +MOVJ EC00076
SMOVL C00077 BC00077 V=166.7  +MOVJ EC00077
SREFP 3 C00078 BC00078  +REFP EC00078
CALL JOB:SEARCH-R1-S13D
SET P021 P006
SFTON3D P021
SMOVL C00079 BC00079 V=166.7  +MOVJ EC00079
SMOVL C00080 BC00080 V=166.7  +MOVJ EC00080
SMOVL C00081 BC00081 V=166.7  +MOVJ EC00081
MOVL C00082 BC00082 V=800.0  +MOVJ EC00082 VJ=100.00
MOVL C00083 BC00083 V=1000.0  +MOVJ EC00083 VJ=100.00
'EndPath S4736
'Path W4732
SFTOF3D
SFTON3D P021
MOVJ C00084 BC00084 VJ=100.00  +MOVJ EC00084 VJ=100.00
SMOVL C00085 BC00085 V=800.0  +MOVJ EC00085
SMOVL C00086 BC00086 V=150.0 PL=0  +MOVJ EC00086
MACRO1 MJ#(0) ARGF14
ARCON
SMOVL C00087 BC00087 V=10.8  +MOVJ EC00087
SMOVL C00088 BC00088 V=11.7  +MOVJ EC00088
SMOVL C00089 BC00089 V=11.7  +MOVJ EC00089
SMOVL C00090 BC00090 V=12.5  +MOVJ EC00090
SMOVL C00091 BC00091 V=12.5  +MOVJ EC00091
SMOVL C00092 BC00092 V=12.5  +MOVJ EC00092
SMOVL C00093 BC00093 V=12.5  +MOVJ EC00093
ARCOF
SMOVL C00094 BC00094 V=800.0  +MOVJ EC00094
SMOVL C00095 BC00095 V=1000.0  +MOVJ EC00095
SFTOF3D
'EndPath W4732
MOVJ C00096 BC00096 VJ=100.00  +MOVJ EC00096 VJ=100.00
MOVJ C00097 BC00097 VJ=100.00  +MOVJ EC00097 VJ=100.00
'Path W4737
SFTOF3D
SFTON3D P022
MOVJ C00098 BC00098 VJ=100.00  +MOVJ EC00098 VJ=100.00
SMOVL C00099 BC00099 V=800.0  +MOVJ EC00099
SMOVL C00100 BC00100 V=150.0 PL=0  +MOVJ EC00100
ARCON
SMOVL C00101 BC00101 V=10.0  +MOVJ EC00101
SMOVL C00102 BC00102 V=10.0  +MOVJ EC00102
ARCOF
SMOVL C00103 BC00103 V=800.0  +MOVJ EC00103
SMOVL C00104 BC00104 V=1000.0  +MOVJ EC00104
SFTOF3D
'EndPath W4737
MOVJ C00105 BC00105 VJ=100.00  +MOVJ EC00105 VJ=100.00
MOVJ C00106 BC00106 VJ=100.00  +MOVJ EC00106 VJ=100.00
'Path W4738
SFTOF3D
SFTON3D P023
MOVJ C00107 BC00107 VJ=100.00  +MOVJ EC00107 VJ=100.00
SMOVL C00108 BC00108 V=800.0  +MOVJ EC00108
SMOVL C00109 BC00109 V=150.0 PL=0  +MOVJ EC00109
ARCON
SMOVL C00110 BC00110 V=10.3  +MOVJ EC00110
SMOVL C00111 BC00111 V=10.3  +MOVJ EC00111
SMOVL C00112 BC00112 V=10.8  +MOVJ EC00112
SFTON3D P024
SMOVL C00113 BC00113 V=10.8  +MOVJ EC00113
SMOVL C00114 BC00114 V=10.8  +MOVJ EC00114
SMOVL C00115 BC00115 V=10.8  +MOVJ EC00115
SMOVL C00116 BC00116 V=10.8  +MOVJ EC00116
SMOVL C00117 BC00117 V=10.8  +MOVJ EC00117
SMOVL C00118 BC00118 V=10.0  +MOVJ EC00118
ARCOF
SMOVL C00119 BC00119 V=800.0  +MOVJ EC00119
SMOVL C00120 BC00120 V=1000.0  +MOVJ EC00120
SFTOF3D
'EndPath W4738
MOVJ C00121 BC00121 VJ=100.00  +MOVJ EC00121 VJ=100.00
MOVJ C00122 BC00122 VJ=100.00  +MOVJ EC00122 VJ=100.00
'Path W4739
SFTOF3D
SFTON3D P025
MOVJ C00123 BC00123 VJ=100.00  +MOVJ EC00123 VJ=100.00
SMOVL C00124 BC00124 V=800.0  +MOVJ EC00124
SMOVL C00125 BC00125 V=150.0 PL=0  +MOVJ EC00125
ARCON
SMOVL C00126 BC00126 V=8.3  +MOVJ EC00126
SMOVL C00127 BC00127 V=8.3  +MOVJ EC00127
ARCOF
SMOVL C00128 BC00128 V=800.0  +MOVJ EC00128
SMOVL C00129 BC00129 V=1000.0  +MOVJ EC00129
SFTOF3D
'EndPath W4739
MOVJ C00130 BC00130 VJ=100.00  +MOVJ EC00130 VJ=100.00
'
MOVJ C00131 BC00131 VJ=100.00  +MOVJ EC00131 VJ=100.00
MOVJ C00132 BC00132 VJ=100.00  +MOVJ EC00132 VJ=100.00
'Path S4745
SFTOF3D
CALL JOB:CLEAN-R1_KM_NEW
MOVJ C00133 BC00133 VJ=100.00  +MOVJ EC00133 VJ=100.00
SFTOF3D
MOVL C00134 BC00134 V=800.0  +MOVJ EC00134 VJ=100.00
SMOVL C00135 BC00135 V=166.7  +MOVJ EC00135
SREFP 3 C00136 BC00136  +REFP EC00136
CALL JOB:SEARCH-R1-S13D
SET P025 P006
SFTON3D P025
SMOVL C00137 BC00137 V=166.7  +MOVJ EC00137
SMOVL C00138 BC00138 V=166.7  +MOVJ EC00138
SREFP 3 C00139 BC00139  +REFP EC00139
CALL JOB:SEARCH-R1-S13D
SET P025 P006
SFTON3D P025
SMOVL C00140 BC00140 V=166.7  +MOVJ EC00140
SMOVL C00141 BC00141 V=166.7  +MOVJ EC00141
SMOVL C00142 BC00142 V=166.7  +MOVJ EC00142
SREFP 3 C00143 BC00143  +REFP EC00143
CALL JOB:SEARCH-R1-S13D
SET P025 P006
SFTON3D P025
SMOVL C00144 BC00144 V=166.7  +MOVJ EC00144
SMOVL C00145 BC00145 V=166.7  +MOVJ EC00145
SMOVL C00146 BC00146 V=166.7  +MOVJ EC00146
MOVL C00147 BC00147 V=800.0  +MOVJ EC00147 VJ=100.00
MOVL C00148 BC00148 V=1000.0  +MOVJ EC00148 VJ=100.00
'EndPath S4745
MOVJ C00149 BC00149 VJ=100.00  +MOVJ EC00149 VJ=100.00
MOVJ C00150 BC00150 VJ=100.00  +MOVJ EC00150 VJ=100.00
'Path S4744
SFTOF3D
MOVJ C00151 BC00151 VJ=100.00  +MOVJ EC00151 VJ=100.00
MOVL C00152 BC00152 V=800.0  +MOVJ EC00152 VJ=100.00
SMOVL C00153 BC00153 V=166.7  +MOVJ EC00153
SREFP 3 C00154 BC00154  +REFP EC00154
CALL JOB:SEARCH-R1-S13D
SET P024 P006
SFTON3D P024
SMOVL C00155 BC00155 V=166.7  +MOVJ EC00155
SMOVL C00156 BC00156 V=166.7  +MOVJ EC00156
SREFP 3 C00157 BC00157  +REFP EC00157
CALL JOB:SEARCH-R1-S13D
SET P024 P006
SFTON3D P024
SMOVL C00158 BC00158 V=166.7  +MOVJ EC00158
SMOVL C00159 BC00159 V=166.7  +MOVJ EC00159
SMOVL C00160 BC00160 V=166.7  +MOVJ EC00160
SREFP 3 C00161 BC00161  +REFP EC00161
CALL JOB:SEARCH-R1-S13D
SET P024 P006
SFTON3D P024
SMOVL C00162 BC00162 V=166.7  +MOVJ EC00162
SMOVL C00163 BC00163 V=166.7  +MOVJ EC00163
SMOVL C00164 BC00164 V=166.7  +MOVJ EC00164
MOVL C00165 BC00165 V=800.0  +MOVJ EC00165 VJ=100.00
MOVL C00166 BC00166 V=1000.0  +MOVJ EC00166 VJ=100.00
'EndPath S4744
MOVJ C00167 BC00167 VJ=100.00  +MOVJ EC00167 VJ=100.00
MOVJ C00168 BC00168 VJ=100.00  +MOVJ EC00168 VJ=100.00
'Path S4743
SFTOF3D
MOVJ C00169 BC00169 VJ=100.00  +MOVJ EC00169 VJ=100.00
MOVL C00170 BC00170 V=800.0  +MOVJ EC00170 VJ=100.00
SMOVL C00171 BC00171 V=166.7  +MOVJ EC00171
SREFP 3 C00172 BC00172  +REFP EC00172
CALL JOB:SEARCH-R1-S13D
SET P023 P006
SFTON3D P023
SMOVL C00173 BC00173 V=166.7  +MOVJ EC00173
SMOVL C00174 BC00174 V=166.7  +MOVJ EC00174
SREFP 3 C00175 BC00175  +REFP EC00175
CALL JOB:SEARCH-R1-S13D
SET P023 P006
SFTON3D P023
SMOVL C00176 BC00176 V=166.7  +MOVJ EC00176
MOVL C00177 BC00177 V=800.0  +MOVJ EC00177 VJ=100.00
MOVL C00178 BC00178 V=1000.0  +MOVJ EC00178 VJ=100.00
'EndPath S4743
MOVJ C00179 BC00179 VJ=100.00  +MOVJ EC00179 VJ=100.00
MOVJ C00180 BC00180 VJ=100.00  +MOVJ EC00180 VJ=100.00
'Path S4742
SFTOF3D
MOVJ C00181 BC00181 VJ=100.00  +MOVJ EC00181 VJ=100.00
MOVL C00182 BC00182 V=800.0  +MOVJ EC00182 VJ=100.00
SMOVL C00183 BC00183 V=166.7  +MOVJ EC00183
SREFP 3 C00184 BC00184  +REFP EC00184
CALL JOB:SEARCH-R1-S13D
SET P022 P006
SFTON3D P022
SMOVL C00185 BC00185 V=166.7  +MOVJ EC00185
SMOVL C00186 BC00186 V=166.7  +MOVJ EC00186
SREFP 3 C00187 BC00187  +REFP EC00187
CALL JOB:SEARCH-R1-S13D
SET P022 P006
SFTON3D P022
SMOVL C00188 BC00188 V=166.7  +MOVJ EC00188
SMOVL C00189 BC00189 V=166.7  +MOVJ EC00189
SMOVL C00190 BC00190 V=166.7  +MOVJ EC00190
SREFP 3 C00191 BC00191  +REFP EC00191
CALL JOB:SEARCH-R1-S13D
SET P022 P006
SFTON3D P022
SMOVL C00192 BC00192 V=166.7  +MOVJ EC00192
SMOVL C00193 BC00193 V=166.7  +MOVJ EC00193
SMOVL C00194 BC00194 V=166.7  +MOVJ EC00194
MOVL C00195 BC00195 V=800.0  +MOVJ EC00195 VJ=100.00
MOVL C00196 BC00196 V=1000.0  +MOVJ EC00196 VJ=100.00
'EndPath S4742
MOVJ C00197 BC00197 VJ=100.00  +MOVJ EC00197 VJ=100.00
MOVJ C00198 BC00198 VJ=100.00  +MOVJ EC00198 VJ=100.00
'Path S4741
SFTOF3D
MOVJ C00199 BC00199 VJ=100.00  +MOVJ EC00199 VJ=100.00
MOVL C00200 BC00200 V=800.0  +MOVJ EC00200 VJ=100.00
SMOVL C00201 BC00201 V=166.7  +MOVJ EC00201
SREFP 3 C00202 BC00202  +REFP EC00202
CALL JOB:SEARCH-R1-S13D
SET P021 P006
SFTON3D P021
SMOVL C00203 BC00203 V=166.7  +MOVJ EC00203
SMOVL C00204 BC00204 V=166.7  +MOVJ EC00204
SREFP 3 C00205 BC00205  +REFP EC00205
CALL JOB:SEARCH-R1-S13D
SET P021 P006
SFTON3D P021
SMOVL C00206 BC00206 V=166.7  +MOVJ EC00206
SMOVL C00207 BC00207 V=166.7  +MOVJ EC00207
SMOVL C00208 BC00208 V=166.7  +MOVJ EC00208
SREFP 3 C00209 BC00209  +REFP EC00209
CALL JOB:SEARCH-R1-S13D
SET P021 P006
SFTON3D P021
SMOVL C00210 BC00210 V=166.7  +MOVJ EC00210
SMOVL C00211 BC00211 V=166.7  +MOVJ EC00211
SMOVL C00212 BC00212 V=166.7  +MOVJ EC00212
MOVL C00213 BC00213 V=800.0  +MOVJ EC00213 VJ=100.00
MOVL C00214 BC00214 V=1000.0  +MOVJ EC00214 VJ=100.00
'EndPath S4741
'Path W4746
SFTOF3D
SFTON3D P021
MOVJ C00215 BC00215 VJ=100.00  +MOVJ EC00215 VJ=100.00
SMOVL C00216 BC00216 V=800.0  +MOVJ EC00216
SMOVL C00217 BC00217 V=150.0 PL=0  +MOVJ EC00217
ARCON
SMOVL C00218 BC00218 V=11.7  +MOVJ EC00218
SMOVL C00219 BC00219 V=11.7  +MOVJ EC00219
SMOVL C00220 BC00220 V=12.5  +MOVJ EC00220
SMOVL C00221 BC00221 V=12.5  +MOVJ EC00221
SMOVL C00222 BC00222 V=12.5  +MOVJ EC00222
SMOVL C00223 BC00223 V=12.5  +MOVJ EC00223
SMOVL C00224 BC00224 V=12.5  +MOVJ EC00224
ARCOF
SMOVL C00225 BC00225 V=800.0  +MOVJ EC00225
SMOVL C00226 BC00226 V=1000.0  +MOVJ EC00226
SFTOF3D
'EndPath W4746
MOVJ C00227 BC00227 VJ=100.00  +MOVJ EC00227 VJ=100.00
MOVJ C00228 BC00228 VJ=100.00  +MOVJ EC00228 VJ=100.00
'Path W4747
SFTOF3D
SFTON3D P022
MOVJ C00229 BC00229 VJ=100.00  +MOVJ EC00229 VJ=100.00
SMOVL C00230 BC00230 V=800.0  +MOVJ EC00230
SMOVL C00231 BC00231 V=150.0 PL=0  +MOVJ EC00231
ARCON
SMOVL C00232 BC00232 V=10.0  +MOVJ EC00232
SMOVL C00233 BC00233 V=10.0  +MOVJ EC00233
SMOVL C00234 BC00234 V=10.0  +MOVJ EC00234
ARCOF
SMOVL C00235 BC00235 V=800.0  +MOVJ EC00235
SMOVL C00236 BC00236 V=1000.0  +MOVJ EC00236
SFTOF3D
'EndPath W4747
MOVJ C00237 BC00237 VJ=100.00  +MOVJ EC00237 VJ=100.00
MOVJ C00238 BC00238 VJ=100.00  +MOVJ EC00238 VJ=100.00
'Path W4748
SFTOF3D
SFTON3D P023
MOVJ C00239 BC00239 VJ=100.00  +MOVJ EC00239 VJ=100.00
SMOVL C00240 BC00240 V=800.0  +MOVJ EC00240
SMOVL C00241 BC00241 V=150.0 PL=0  +MOVJ EC00241
ARCON
SMOVL C00242 BC00242 V=10.0  +MOVJ EC00242
SMOVL C00243 BC00243 V=10.0  +MOVJ EC00243
SMOVL C00244 BC00244 V=10.8  +MOVJ EC00244
SFTON3D P024
SMOVL C00245 BC00245 V=10.8  +MOVJ EC00245
SMOVL C00246 BC00246 V=10.8  +MOVJ EC00246
SMOVL C00247 BC00247 V=10.8  +MOVJ EC00247
SMOVL C00248 BC00248 V=10.8  +MOVJ EC00248
SMOVL C00249 BC00249 V=10.0  +MOVJ EC00249
SMOVL C00250 BC00250 V=10.0  +MOVJ EC00250
ARCOF
SMOVL C00251 BC00251 V=800.0  +MOVJ EC00251
SMOVL C00252 BC00252 V=1000.0  +MOVJ EC00252
SFTOF3D
'EndPath W4748
MOVJ C00253 BC00253 VJ=100.00  +MOVJ EC00253 VJ=100.00
MOVJ C00254 BC00254 VJ=100.00  +MOVJ EC00254 VJ=100.00
'Path W4749
SFTOF3D
SFTON3D P025
MOVJ C00255 BC00255 VJ=100.00  +MOVJ EC00255 VJ=100.00
SMOVL C00256 BC00256 V=800.0  +MOVJ EC00256
SMOVL C00257 BC00257 V=150.0 PL=0  +MOVJ EC00257
ARCON
SMOVL C00258 BC00258 V=9.2  +MOVJ EC00258
SMOVL C00259 BC00259 V=9.2  +MOVJ EC00259
ARCOF
SMOVL C00260 BC00260 V=800.0  +MOVJ EC00260
SMOVL C00261 BC00261 V=1000.0  +MOVJ EC00261
SFTOF3D
'EndPath W4749
MOVJ C00262 BC00262 VJ=100.00  +MOVJ EC00262 VJ=100.00
MOVJ C00263 BC00263 VJ=100.00  +MOVJ EC00263 VJ=100.00
MOVJ C00264 BC00264 VJ=100.00  +MOVJ EC00264 VJ=100.00
CALL JOB:CLEAN-R1_KM_NEW
'
'
'
MOVJ C00265 BC00265 VJ=100.00  +MOVJ EC00265 VJ=100.00
'Path S4750
SFTOF3D
MOVJ C00266 BC00266 VJ=100.00  +MOVJ EC00266 VJ=100.00
MOVL C00267 BC00267 V=800.0  +MOVJ EC00267 VJ=100.00
SMOVL C00268 BC00268 V=166.7  +MOVJ EC00268
SREFP 3 C00269 BC00269  +REFP EC00269
CALL JOB:SEARCH-R1-S13D
SET P035 P006
SFTON3D P035
SMOVL C00270 BC00270 V=166.7  +MOVJ EC00270
SMOVL C00271 BC00271 V=166.7  +MOVJ EC00271
SREFP 3 C00272 BC00272  +REFP EC00272
CALL JOB:SEARCH-R1-S13D
SET P035 P006
SFTON3D P035
SMOVL C00273 BC00273 V=166.7  +MOVJ EC00273
SMOVL C00274 BC00274 V=166.7  +MOVJ EC00274
SREFP 3 C00275 BC00275  +REFP EC00275
CALL JOB:SEARCH-R1-S13D
SET P035 P006
SFTON3D P035
SMOVL C00276 BC00276 V=166.7  +MOVJ EC00276
MOVL C00277 BC00277 V=800.0  +MOVJ EC00277 VJ=100.00
MOVL C00278 BC00278 V=1000.0  +MOVJ EC00278 VJ=100.00
'EndPath S4750
'Path S4751
SFTOF3D
MOVJ C00279 BC00279 VJ=100.00  +MOVJ EC00279 VJ=100.00
MOVL C00280 BC00280 V=800.0  +MOVJ EC00280 VJ=100.00
SMOVL C00281 BC00281 V=166.7  +MOVJ EC00281
SREFP 3 C00282 BC00282  +REFP EC00282
CALL JOB:SEARCH-R1-S13D
SET P034 P006
SFTON3D P034
SMOVL C00283 BC00283 V=166.7  +MOVJ EC00283
SMOVL C00284 BC00284 V=166.7  +MOVJ EC00284
SREFP 3 C00285 BC00285  +REFP EC00285
CALL JOB:SEARCH-R1-S13D
SET P034 P006
SFTON3D P034
SMOVL C00286 BC00286 V=166.7  +MOVJ EC00286
MOVL C00287 BC00287 V=800.0  +MOVJ EC00287 VJ=100.00
MOVL C00288 BC00288 V=1000.0  +MOVJ EC00288 VJ=100.00
'EndPath S4751
'Path S4752
SFTOF3D
MOVJ C00289 BC00289 VJ=100.00  +MOVJ EC00289 VJ=100.00
MOVL C00290 BC00290 V=800.0  +MOVJ EC00290 VJ=100.00
SMOVL C00291 BC00291 V=166.7  +MOVJ EC00291
SREFP 3 C00292 BC00292  +REFP EC00292
CALL JOB:SEARCH-R1-S13D
SET P033 P006
SFTON3D P033
SMOVL C00293 BC00293 V=166.7  +MOVJ EC00293
SMOVL C00294 BC00294 V=166.7  +MOVJ EC00294
SREFP 3 C00295 BC00295  +REFP EC00295
CALL JOB:SEARCH-R1-S13D
SET P033 P006
SFTON3D P033
SMOVL C00296 BC00296 V=166.7  +MOVJ EC00296
MOVL C00297 BC00297 V=800.0  +MOVJ EC00297 VJ=100.00
MOVL C00298 BC00298 V=1000.0  +MOVJ EC00298 VJ=100.00
'EndPath S4752
'Path S4753
SFTOF3D
MOVJ C00299 BC00299 VJ=100.00  +MOVJ EC00299 VJ=100.00
MOVL C00300 BC00300 V=800.0  +MOVJ EC00300 VJ=100.00
SMOVL C00301 BC00301 V=166.7  +MOVJ EC00301
SREFP 3 C00302 BC00302  +REFP EC00302
CALL JOB:SEARCH-R1-S13D
SET P032 P006
SFTON3D P032
SMOVL C00303 BC00303 V=166.7  +MOVJ EC00303
SMOVL C00304 BC00304 V=166.7  +MOVJ EC00304
SREFP 3 C00305 BC00305  +REFP EC00305
CALL JOB:SEARCH-R1-S13D
SET P032 P006
SFTON3D P032
SMOVL C00306 BC00306 V=166.7  +MOVJ EC00306
MOVL C00307 BC00307 V=800.0  +MOVJ EC00307 VJ=100.00
MOVL C00308 BC00308 V=1000.0  +MOVJ EC00308 VJ=100.00
'EndPath S4753
'Path S4754
SFTOF3D
MOVJ C00309 BC00309 VJ=100.00  +MOVJ EC00309 VJ=100.00
MOVL C00310 BC00310 V=800.0  +MOVJ EC00310 VJ=100.00
SMOVL C00311 BC00311 V=166.7  +MOVJ EC00311
SREFP 3 C00312 BC00312  +REFP EC00312
CALL JOB:SEARCH-R1-S13D
SET P032 P006
SFTON3D P032
SMOVL C00313 BC00313 V=166.7  +MOVJ EC00313
SMOVL C00314 BC00314 V=166.7  +MOVJ EC00314
SREFP 3 C00315 BC00315  +REFP EC00315
CALL JOB:SEARCH-R1-S13D
SET P032 P006
SFTON3D P032
SMOVL C00316 BC00316 V=166.7  +MOVJ EC00316
MOVL C00317 BC00317 V=800.0  +MOVJ EC00317 VJ=100.00
MOVL C00318 BC00318 V=1000.0  +MOVJ EC00318 VJ=100.00
'EndPath S4754
'Path S4756
SFTOF3D
MOVJ C00319 BC00319 VJ=100.00  +MOVJ EC00319 VJ=100.00
MOVL C00320 BC00320 V=800.0  +MOVJ EC00320 VJ=100.00
SMOVL C00321 BC00321 V=166.7  +MOVJ EC00321
SREFP 3 C00322 BC00322  +REFP EC00322
CALL JOB:SEARCH-R1-S13D
SET P031 P006
SFTON3D P031
SMOVL C00323 BC00323 V=166.7  +MOVJ EC00323
SMOVL C00324 BC00324 V=166.7  +MOVJ EC00324
SREFP 3 C00325 BC00325  +REFP EC00325
CALL JOB:SEARCH-R1-S13D
SET P031 P006
SFTON3D P031
SMOVL C00326 BC00326 V=166.7  +MOVJ EC00326
SMOVL C00327 BC00327 V=166.7  +MOVJ EC00327
SREFP 3 C00328 BC00328  +REFP EC00328
CALL JOB:SEARCH-R1-S13D
SET P031 P006
SFTON3D P031
SMOVL C00329 BC00329 V=166.7  +MOVJ EC00329
MOVL C00330 BC00330 V=800.0  +MOVJ EC00330 VJ=100.00
MOVL C00331 BC00331 V=1000.0  +MOVJ EC00331 VJ=100.00
'EndPath S4756
'Path W4751
SFTOF3D
SFTON3D P032
MOVJ C00332 BC00332 VJ=100.00  +MOVJ EC00332 VJ=100.00
SMOVL C00333 BC00333 V=800.0  +MOVJ EC00333
SMOVL C00334 BC00334 V=150.0 PL=0  +MOVJ EC00334
MACRO1 MJ#(0) ARGF21
ARCON
SFTON3D P031
SMOVL C00335 BC00335 V=7.5  +MOVJ EC00335
SMOVL C00336 BC00336 V=7.5  +MOVJ EC00336
ARCOF
SMOVL C00337 BC00337 V=800.0  +MOVJ EC00337
SMOVL C00338 BC00338 V=1000.0  +MOVJ EC00338
SFTOF3D
'EndPath W4751
'Path W4755
SFTOF3D
SFTON3D P034
MOVJ C00339 BC00339 VJ=100.00  +MOVJ EC00339 VJ=100.00
SMOVL C00340 BC00340 V=800.0  +MOVJ EC00340
SMOVL C00341 BC00341 V=150.0 PL=0  +MOVJ EC00341
ARCON
SFTON3D P035
SMOVL C00342 BC00342 V=7.5  +MOVJ EC00342
SMOVL C00343 BC00343 V=7.5  +MOVJ EC00343
ARCOF
SMOVL C00344 BC00344 V=800.0  +MOVJ EC00344
SMOVL C00345 BC00345 V=1000.0  +MOVJ EC00345
SFTOF3D
'EndPath W4755
'Path W4752
SFTOF3D
SFTON3D P032
MOVJ C00346 BC00346 VJ=100.00  +MOVJ EC00346 VJ=100.00
SMOVL C00347 BC00347 V=800.0  +MOVJ EC00347
SMOVL C00348 BC00348 V=150.0 PL=0  +MOVJ EC00348
ARCON
SFTON3D P033
SMOVL C00349 BC00349 V=7.5  +MOVJ EC00349
ARCOF
SMOVL C00350 BC00350 V=800.0  +MOVJ EC00350
SMOVL C00351 BC00351 V=1000.0  +MOVJ EC00351
SFTOF3D
'EndPath W4752
'Path W4754
SFTOF3D
SFTON3D P034
MOVJ C00352 BC00352 VJ=100.00  +MOVJ EC00352 VJ=100.00
SMOVL C00353 BC00353 V=800.0  +MOVJ EC00353
SMOVL C00354 BC00354 V=150.0 PL=0  +MOVJ EC00354
ARCON
SFTON3D P033
SMOVL C00355 BC00355 V=8.3  +MOVJ EC00355
SMOVL C00356 BC00356 V=8.3  +MOVJ EC00356
ARCOF
SMOVL C00357 BC00357 V=800.0  +MOVJ EC00357
SMOVL C00358 BC00358 V=1000.0  +MOVJ EC00358
SFTOF3D
SMOVL C00359 BC00359 V=1000.0  +MOVJ EC00359
SMOVL C00360 BC00360 V=1000.0  +MOVJ EC00360
SMOVL C00361 BC00361 V=1000.0  +MOVJ EC00361
SMOVL C00362 BC00362 V=1000.0  +MOVJ EC00362
SMOVL C00363 BC00363 V=250.0  +MOVJ EC00363
ARCON
SMOVL C00364 BC00364 V=8.3  +MOVJ EC00364
SFTON3D P031
SMOVL C00365 BC00365 V=8.3  +MOVJ EC00365
ARCOF
SMOVL C00366 BC00366 V=250.0  +MOVJ EC00366
SMOVL C00367 BC00367 V=250.0  +MOVJ EC00367
SMOVL C00368 BC00368 V=250.0  +MOVJ EC00368
SMOVL C00369 BC00369 V=250.0  +MOVJ EC00369
ARCON
SMOVL C00370 BC00370 V=8.3  +MOVJ EC00370
SMOVL C00371 BC00371 V=8.3  +MOVJ EC00371
ARCOF
SMOVL C00372 BC00372 V=250.0  +MOVJ EC00372
SFTOF3D
'EndPath W4754
MOVJ C00373 BC00373 VJ=100.00  +MOVJ EC00373 VJ=100.00
MOVJ C00374 BC00374 VJ=100.00  +MOVJ EC00374 VJ=100.00
MOVJ C00375 BC00375 VJ=100.00  +MOVJ EC00375 VJ=100.00
MOVJ C00376 BC00376 VJ=15.00  +MOVJ EC00376 VJ=100.00
SFTON3D P035
SMOVL C00377 BC00377 V=166.7  +MOVJ EC00377
ARCON
SMOVL C00378 BC00378 V=8.3  +MOVJ EC00378
SMOVL C00379 BC00379 V=8.3  +MOVJ EC00379
SMOVL C00380 BC00380 V=8.3  +MOVJ EC00380
ARCOF
MOVJ C00381 BC00381 VJ=100.00  +MOVJ EC00381 VJ=100.00
MOVJ C00382 BC00382 VJ=100.00  +MOVJ EC00382 VJ=100.00
SMOVL C00383 BC00383 V=166.7  +MOVJ EC00383
ARCON
SMOVL C00384 BC00384 V=7.5  +MOVJ EC00384
SMOVL C00385 BC00385 V=7.5  +MOVJ EC00385
ARCOF
SMOVL C00386 BC00386 V=166.7  +MOVJ EC00386
SMOVL C00387 BC00387 V=166.7  +MOVJ EC00387
SFTOF3D
MOVJ C00388 BC00388 VJ=100.00  +MOVJ EC00388 VJ=100.00
MOVJ C00389 BC00389 VJ=100.00  +MOVJ EC00389 VJ=100.00
END
